SUBAPPLICATION ManyOutputsSIFB025 (* Subapplication Type *)
  (* Standard: 61499-2 *)
  (* Version 1.0, 2025-05-03, cochicde *)
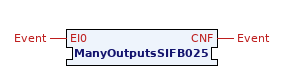
  EVENT_INPUT
    EI0;
  END_EVENT
  EVENT_OUTPUT
    CNF;
  END_EVENT
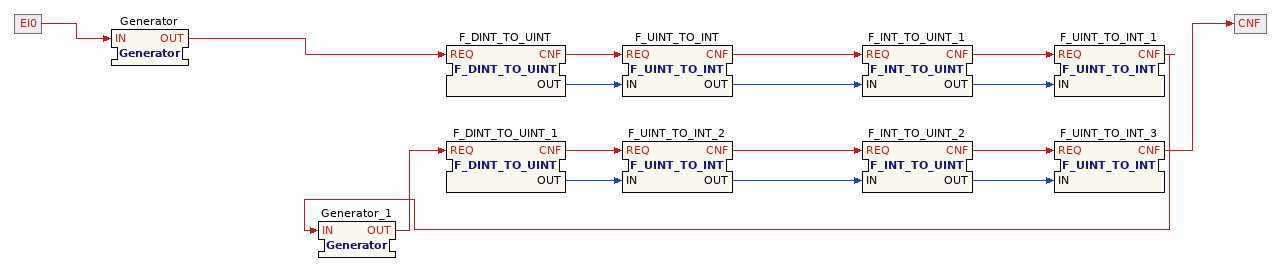
  FBS
    F_DINT_TO_UINT : F_DINT_TO_UINT;
    Generator_1 : performance::Generator;
    F_INT_TO_UINT_1 : F_INT_TO_UINT;
    F_INT_TO_UINT_2 : F_INT_TO_UINT;
    Generator : performance::Generator;
    F_UINT_TO_INT_2 : F_UINT_TO_INT;
    F_DINT_TO_UINT_1 : F_DINT_TO_UINT;
    F_UINT_TO_INT_1 : F_UINT_TO_INT;
    F_UINT_TO_INT : F_UINT_TO_INT;
    F_UINT_TO_INT_3 : F_UINT_TO_INT;
  END_FBS
  EVENT_CONNECTIONS
    Generator.OUT TO F_DINT_TO_UINT.REQ;
    F_DINT_TO_UINT.CNF TO F_UINT_TO_INT.REQ;
    Generator_1.OUT TO F_DINT_TO_UINT_1.REQ;
    F_UINT_TO_INT.CNF TO F_INT_TO_UINT_1.REQ;
    F_INT_TO_UINT_1.CNF TO F_UINT_TO_INT_1.REQ;
    F_UINT_TO_INT_2.CNF TO F_INT_TO_UINT_2.REQ;
    F_INT_TO_UINT_2.CNF TO F_UINT_TO_INT_3.REQ;
    F_DINT_TO_UINT_1.CNF TO F_UINT_TO_INT_2.REQ;
    F_UINT_TO_INT_1.CNF TO Generator_1.IN;
    F_UINT_TO_INT_3.CNF TO CNF;
    EI0 TO Generator.IN;
  END_CONNECTIONS
  DATA_CONNECTIONS
    F_DINT_TO_UINT.OUT TO F_UINT_TO_INT.IN;
    F_UINT_TO_INT.OUT TO F_INT_TO_UINT_1.IN;
    F_INT_TO_UINT_1.OUT TO F_UINT_TO_INT_1.IN;
    F_UINT_TO_INT_2.OUT TO F_INT_TO_UINT_2.IN;
    F_INT_TO_UINT_2.OUT TO F_UINT_TO_INT_3.IN;
    F_DINT_TO_UINT_1.OUT TO F_UINT_TO_INT_2.IN;
  END_CONNECTIONS
END_SUBAPPLICATION
